FUNCTION_BLOCK FB_DataHistory_Int
VAR_INPUT
	_val : INT;
	_save : BOOL;
END_VAR
VAR_OUTPUT
	_array : ARRAY [0..DatenHistoryZaehler] OF INT;
END_VAR
VAR
	_i : INT;
END_VAR

IF _save THEN
	FOR _i := 0 TO DatenHistoryZaehler - 1 DO
		_array[_i] := _array[_i + 1];
	END_FOR
	_array[DatenHistoryZaehler] := _val;
END_IF

END_FUNCTION_BLOCK

(* stored: Version 1.1.0.1, ProductVersion 3.1.4018.5
   POU FB_DataHistory_Int: Id {680c2198-cf2d-440e-8929-654d1bad9ca6}, SpecialFunc None *)
